INTERFACE I_XP_Path  EXTENDS __SYSTEM.IQueryInterface, I_CH_Object

METHOD DistanceToDestiantion : LREAL
VAR_INPUT
	ipTrack : I_XP_Track;
	fPosOnTrack : LREAL;
END_VAR
END_METHOD

{attribute 'monitoring':='call'}
PROPERTY Length : LREAL
GET
END_GET
SET
END_SET
END_PROPERTY

PROPERTY PointerToThis : POINTER TO FB_XP_Path
GET
END_GET
END_PROPERTY

{attribute 'monitoring':='call'}
PROPERTY StationDestination : I_XP_Station
GET
END_GET
SET
END_SET
END_PROPERTY

{attribute 'monitoring':='call'}
PROPERTY StationStart  : I_XP_Station
GET
END_GET
SET
END_SET
END_PROPERTY

{attribute 'monitoring':='call'}
PROPERTY TracksUsed : REFERENCE TO FB_CH_List
GET
END_GET
END_PROPERTY

END_INTERFACE

(* stored: Version 1.1.0.1, ProductVersion 3.1.4024.12
   Itf I_XP_Path: Id {d0a7e409-20e8-490f-be78-3b4ffcbf57b0}
   Method DistanceToDestiantion: Id {16fcaeeb-05bd-43dc-9bde-b5fbe4442f30}
   Property Length: Id {cb708bc0-0881-4fe2-948c-5f52e598f6b1}
   Get Get: Id {30585cc5-fce9-4484-9065-89d0cda9ba65}
   Set Set: Id {e5b36e72-b398-44b3-b515-7e84f3c44be8}
   Property PointerToThis: Id {2dd54737-87ff-403b-bec1-2c19dbbf8181}
   Get Get: Id {31b8df92-0c58-4bb2-aecd-e42541e7fbef}
   Property StationDestination: Id {0b1ccaa1-9c39-4bc1-b84e-444daddcdd93}
   Get Get: Id {07455a68-e4cc-4252-8dca-847b5ac55671}
   Set Set: Id {907b8bc7-e7be-4ea3-8475-481a6af30df2}
   Property StationStart: Id {6e510288-2b3b-4ba7-8b21-f3421a7b860b}
   Get Get: Id {ed5754e4-4b4c-4ec1-a307-000d48e50e38}
   Set Set: Id {3c398c49-dfe3-4d3b-955a-2dd846681446}
   Property TracksUsed: Id {016f7596-979f-4883-a183-27b80a0716c6}
   Get Get: Id {5387341d-8ab0-4f96-a112-1a35ae044f5f} *)
